Universal Robots PolyScope program: ControlReset.urp

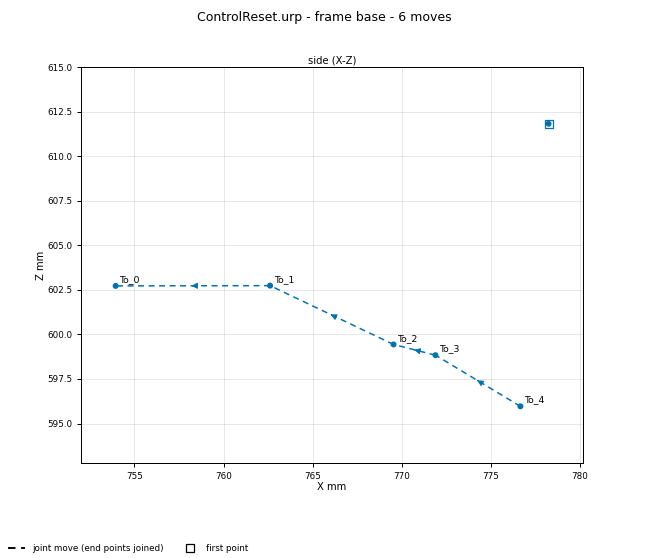
[picture p0: tool path of ControlReset.urp in frame base, 6 of 9 moves have a stored position in this frame; points joined in program order, loops and branches not executed]
Program ControlReset (installation=Youssef directory=/programs/Youssef createdIn=5.9.5.1031259 lastSavedIn=5.9.5.1031259 robotSerialNumber=20215500597)
Calibrated DH parameters: a=[0.000193, -0.066673, -0.391568, -0.000012, 0.00005, 0]; d=[0.162643, -472.05677, 465.132521, 7.058239, 0.099746, 0.099582]; alpha=[1.571116, 0.00089, 0.003862, 1.569269, -1.569248, 0]; deltaTheta=[0, -1.413394, 7.628392, 0.068187, 0, -0.000001]
Robot Program (runOnlyOnce=true)
  MoveJ speed 60 deg/s, acceleration 80 deg/s^2 (useActiveTCP=true) feature=Base
    Waypoint Waypoint (Variable): variable(featureName=Control_Standby)
    Waypoint Waypoint_3: TCP in base x=778.24 y=-17.942 z=611.823 mm, rx=-0.0636 ry=2.4704 rz=-0.2743 rad; joints [170.473, -63.159, 27.038, -93.122, -94.218, 75.99] deg; TCP offset x=0 y=0 z=191.5 mm, rx=0 ry=0 rz=0 rad
    Waypoint Waypoint (Variable): variable(featureName=Control_R_End)
    Waypoint To_4: motionParameters(jointSpeed=1.047198 jointAcceleration=1.396263 cartesianSpeed=0.1 cartesianAcceleration=1.2); TCP in base x=776.661 y=-17.794 z=595.965 mm, rx=-0.0637 ry=2.4705 rz=-0.2742 rad; joints [170.456, -65.851, 34.031, -97.42, -94.206, 75.991] deg
    Waypoint To_3: motionParameters(jointSpeed=1.047198 jointAcceleration=1.396263 cartesianSpeed=0.1 cartesianAcceleration=1.2); TCP in base x=771.893 y=-17.795 z=598.835 mm, rx=-0.0637 ry=2.4705 rz=-0.2742 rad; joints [170.378, -66.476, 34.483, -97.248, -94.158, 75.93] deg
    Waypoint To_2: motionParameters(jointSpeed=1.047198 jointAcceleration=1.396263 cartesianSpeed=0.1 cartesianAcceleration=1.2); TCP in base x=769.54 y=-17.783 z=599.437 mm, rx=-0.0638 ry=2.4705 rz=-0.2742 rad; joints [170.339, -66.884, 34.994, -97.353, -94.131, 75.897] deg
    Waypoint To_1: motionParameters(jointSpeed=1.047198 jointAcceleration=1.396263 cartesianSpeed=0.1 cartesianAcceleration=1.2); TCP in base x=762.609 y=-17.768 z=602.737 mm, rx=-0.0638 ry=2.4705 rz=-0.2742 rad; joints [170.223, -67.881, 35.915, -97.286, -94.059, 75.807] deg
    Waypoint To_0: motionParameters(jointSpeed=1.047198 jointAcceleration=1.396263 cartesianSpeed=0.1 cartesianAcceleration=1.2); TCP in base x=753.941 y=-17.776 z=602.724 mm, rx=-0.0637 ry=2.4705 rz=-0.2742 rad; joints [170.071, -69.568, 38.384, -98.074, -93.963, 75.694] deg
    Waypoint Waypoint (Variable): variable(featureName=Control_Standby)
